{attribute 'qualified_only'}
VAR_GLOBAL
	testBoolLinker : BOOL := FALSE;
	testBoolLinker2 : BOOL := FALSE;
END_VAR

(* stored: Version 1.1.0.1
   GVL test: Id {a1ba38c3-67d8-44ae-8a3c-acff49e84665} *)
